TYPE ST_MV_JAVA_Parameter :
STRUCT
	Temp_Heisswasser        : REAL;
	Temp_Heisswasser_Max    : REAL;
	Temp_Heisswasser_Min    : REAL;

END_STRUCT
END_TYPE

(* stored: Version 1.1.0.1, ProductVersion 3.1.4024.9
   DUT ST_MV_JAVA_Parameter: Id {b507bfef-a0ca-4e57-9b9f-a1fbde805354} *)
